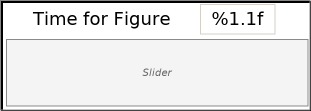
VISUALIZATION InputNumSlider_Time  // 311x111
VAR_IN_OUT
number : REAL;
END_VAR
    Rectangle (1,1 310x110)
    Slider (6,39 302x67), variable: number, scale 0..100
    Textfield (30,4 150x30), "Time for Figure"
    Textfield (200,4 75x30), "%1.1f", text variable: number
        OnMouseClick: write the text variable via Default, min 0, max 360
END_VISUALIZATION

(* stored: Version 1.1.0.1, ProductVersion 3.1.4024.12
   Visu InputNumSlider_Time: Id {dc91846d-02bd-49f4-a028-0fa496a588a8} *)
